// Mitsubishi GX Works2 project: ducthanh   PLC: FX2N/FX2NC

PROGRAM MAIN
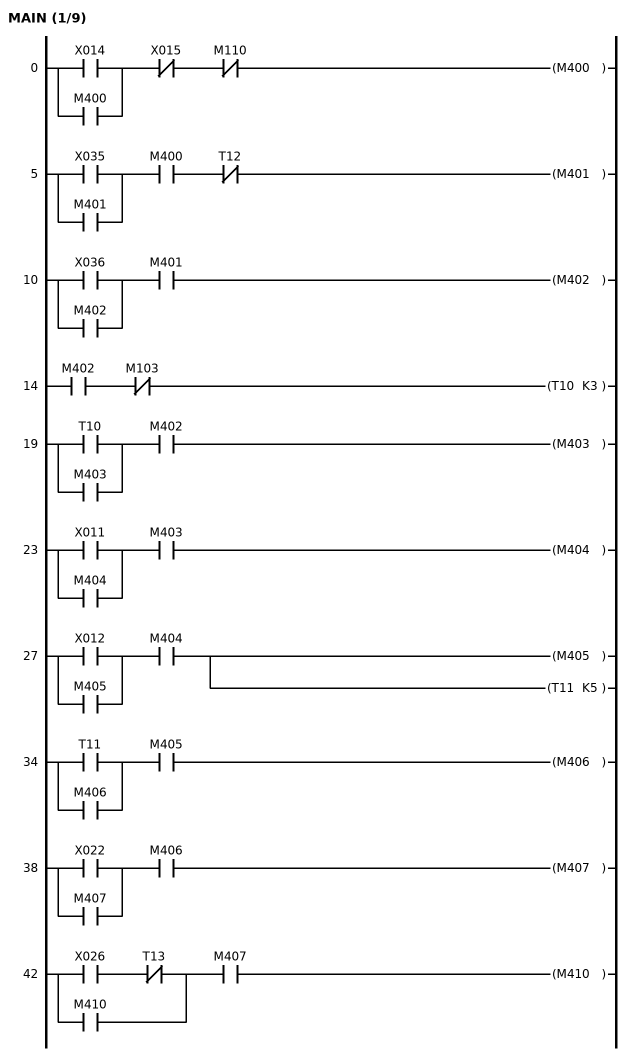
0     LD      X014
      OR      M400
      ANI     X015
      ANI     M110
      OUT     M400
5     LD      X035
      OR      M401
      AND     M400
      ANI     T12
      OUT     M401
10    LD      X036
      OR      M402
      AND     M401
      OUT     M402
14    LD      M402
      ANI     M103
      OUT     T10 K3
19    LD      T10
      OR      M403
      AND     M402
      OUT     M403
23    LD      X011
      OR      M404
      AND     M403
      OUT     M404
27    LD      X012
      OR      M405
      AND     M404
      OUT     M405
      OUT     T11 K5
34    LD      T11
      OR      M406
      AND     M405
      OUT     M406
38    LD      X022
      OR      M407
      AND     M406
      OUT     M407
42    LD      X026
      ANI     T13
      OR      M410
      AND     M407
      OUT     M410
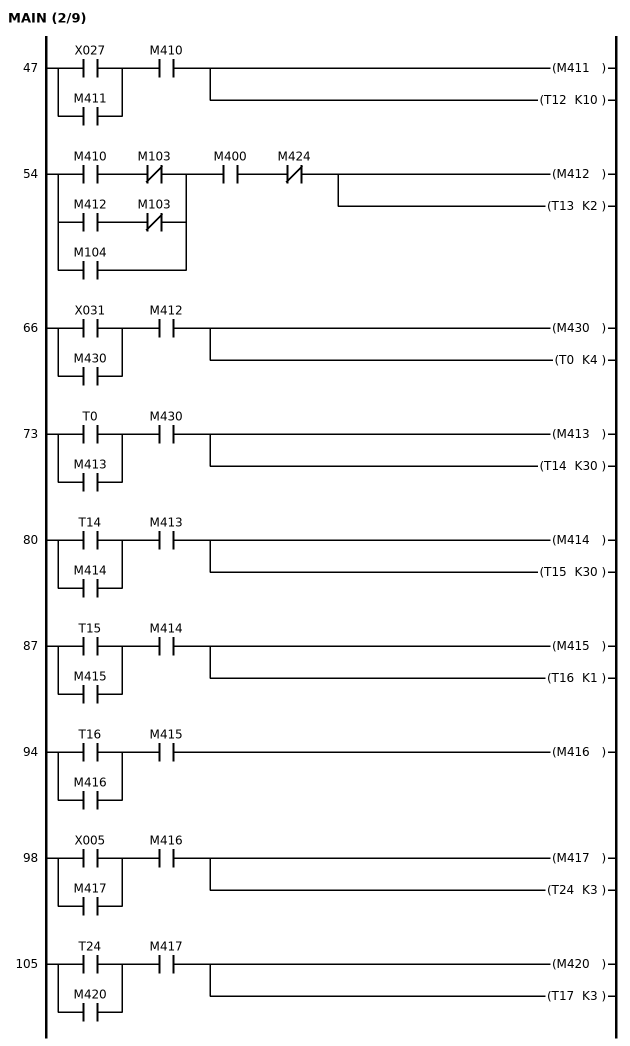
47    LD      X027
      OR      M411
      AND     M410
      OUT     M411
      OUT     T12 K10
54    LD      M410
      ANI     M103
      LD      M412
      ANI     M103
      ORB
      OR      M104
      AND     M400
      ANI     M424
      OUT     M412
      OUT     T13 K2
66    LD      X031
      OR      M430
      AND     M412
      OUT     M430
      OUT     T0 K4
73    LD      T0
      OR      M413
      AND     M430
      OUT     M413
      OUT     T14 K30
80    LD      T14
      OR      M414
      AND     M413
      OUT     M414
      OUT     T15 K30
87    LD      T15
      OR      M415
      AND     M414
      OUT     M415
      OUT     T16 K1
94    LD      T16
      OR      M416
      AND     M415
      OUT     M416
98    LD      X005
      OR      M417
      AND     M416
      OUT     M417
      OUT     T24 K3
105   LD      T24
      OR      M420
      AND     M417
      OUT     M420
      OUT     T17 K3
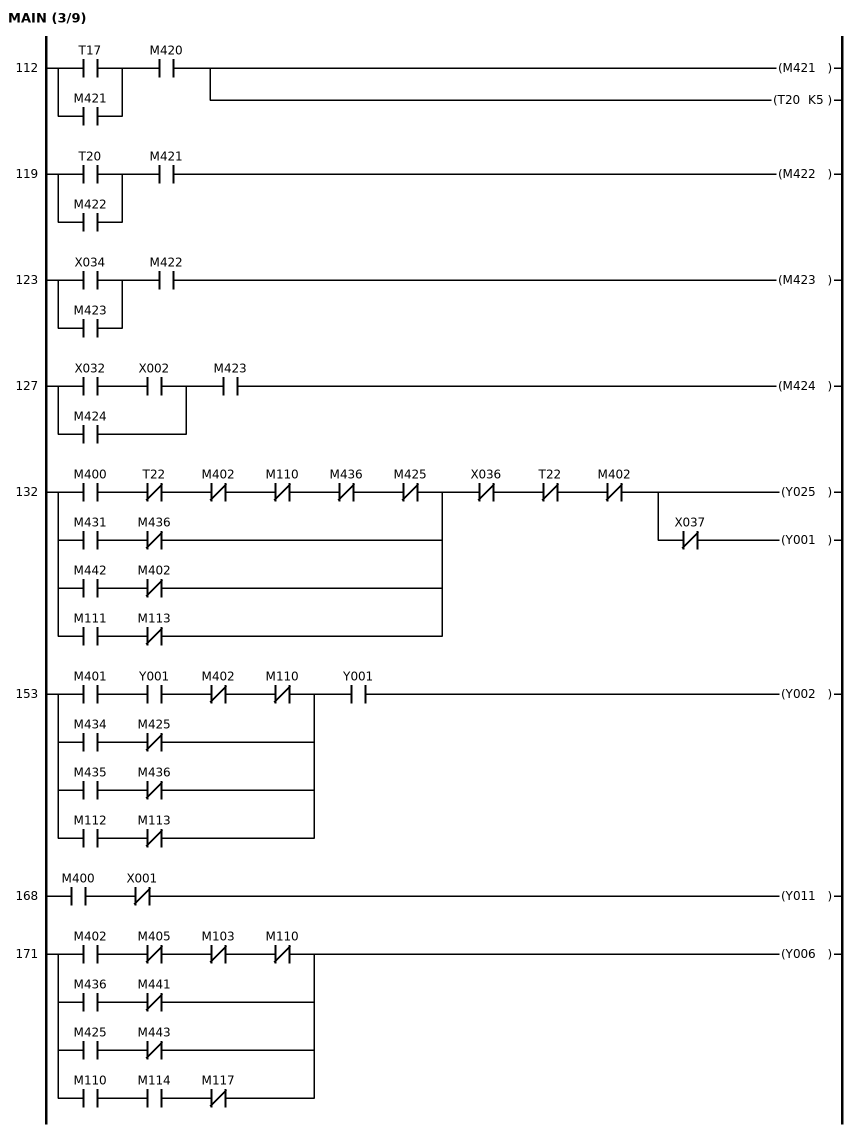
112   LD      T17
      OR      M421
      AND     M420
      OUT     M421
      OUT     T20 K5
119   LD      T20
      OR      M422
      AND     M421
      OUT     M422
123   LD      X034
      OR      M423
      AND     M422
      OUT     M423
127   LD      X032
      AND     X002
      OR      M424
      AND     M423
      OUT     M424
132   LD      M400
      ANI     T22
      ANI     M402
      ANI     M110
      ANI     M436
      ANI     M425
      LD      M431
      ANI     M436
      ORB
      LD      M442
      ANI     M402
      ORB
      LD      M111
      ANI     M113
      ORB
      ANI     X036
      ANI     T22
      ANI     M402
      OUT     Y025
      ANI     X037
      OUT     Y001
153   LD      M401
      AND     Y001
      ANI     M402
      ANI     M110
      LD      M434
      ANI     M425
      ORB
      LD      M435
      ANI     M436
      ORB
      LD      M112
      ANI     M113
      ORB
      AND     Y001
      OUT     Y002
168   LD      M400
      ANI     X001
      OUT     Y011
171   LD      M402
      ANI     M405
      ANI     M103
      ANI     M110
      LD      M436
      ANI     M441
      ORB
      LD      M425
      ANI     M443
      ORB
      LD      M110
      AND     M114
      ANI     M117
      ORB
      OUT     Y006
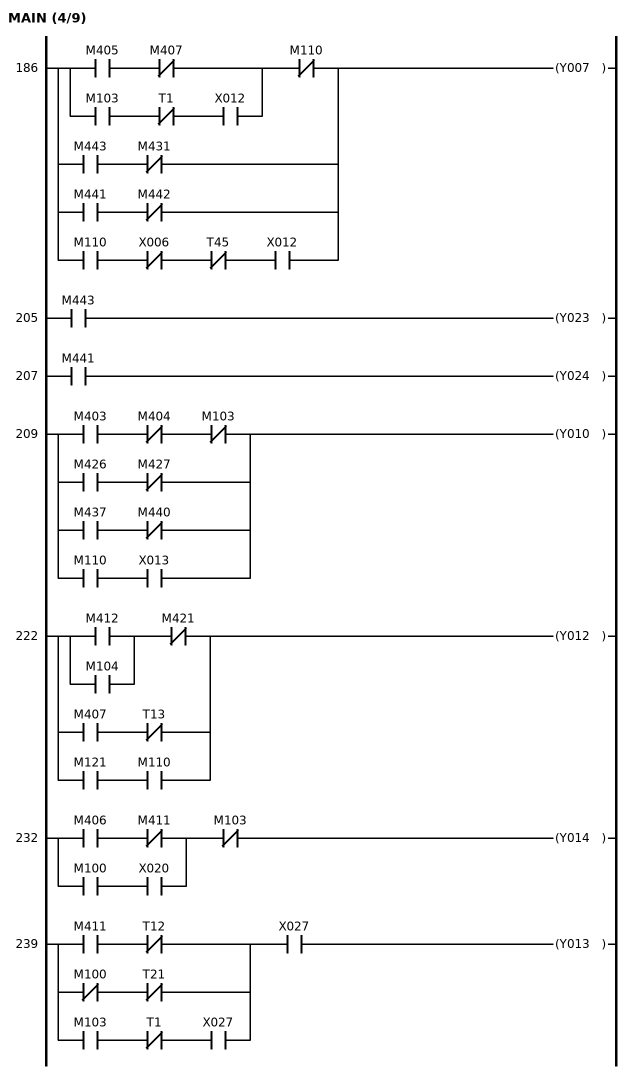
186   LD      M405
      ANI     M407
      LD      M103
      ANI     T1
      AND     X012
      ORB
      ANI     M110
      LD      M443
      ANI     M431
      ORB
      LD      M441
      ANI     M442
      ORB
      LD      M110
      ANI     X006
      ANI     T45
      AND     X012
      ORB
      OUT     Y007
205   LD      M443
      OUT     Y023
207   LD      M441
      OUT     Y024
209   LD      M403
      ANI     M404
      ANI     M103
      LD      M426
      ANI     M427
      ORB
      LD      M437
      ANI     M440
      ORB
      LD      M110
      AND     X013
      ORB
      OUT     Y010
222   LD      M412
      OR      M104
      ANI     M421
      LD      M407
      ANI     T13
      ORB
      LD      M121
      AND     M110
      ORB
      OUT     Y012
232   LD      M406
      ANI     M411
      LD      M100
      AND     X020
      ORB
      ANI     M103
      OUT     Y014
239   LD      M411
      ANI     T12
      LDI     M100
      ANI     T21
      ORB
      LD      M103
      ANI     T1
      AND     X027
      ORB
      AND     X027
      OUT     Y013
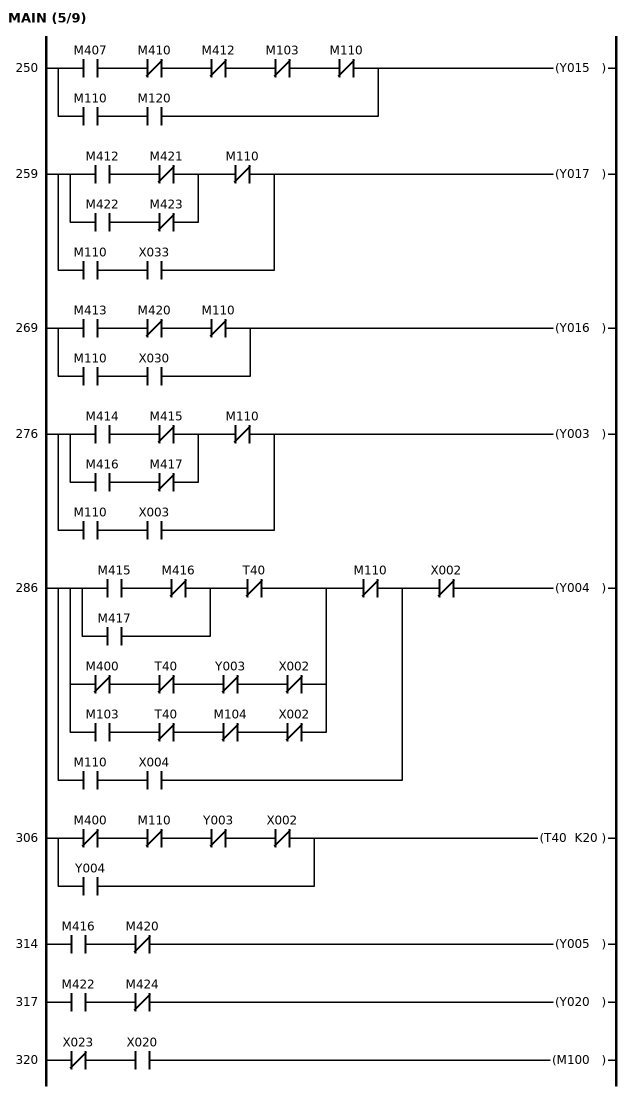
250   LD      M407
      ANI     M410
      ANI     M412
      ANI     M103
      ANI     M110
      LD      M110
      AND     M120
      ORB
      OUT     Y015
259   LD      M412
      ANI     M421
      LD      M422
      ANI     M423
      ORB
      ANI     M110
      LD      M110
      AND     X033
      ORB
      OUT     Y017
269   LD      M413
      ANI     M420
      ANI     M110
      LD      M110
      AND     X030
      ORB
      OUT     Y016
276   LD      M414
      ANI     M415
      LD      M416
      ANI     M417
      ORB
      ANI     M110
      LD      M110
      AND     X003
      ORB
      OUT     Y003
286   LD      M415
      ANI     M416
      OR      M417
      ANI     T40
      LDI     M400
      ANI     T40
      ANI     Y003
      ANI     X002
      ORB
      LD      M103
      ANI     T40
      ANI     M104
      ANI     X002
      ORB
      ANI     M110
      LD      M110
      AND     X004
      ORB
      ANI     X002
      OUT     Y004
306   LDI     M400
      ANI     M110
      ANI     Y003
      ANI     X002
      OR      Y004
      OUT     T40 K20
314   LD      M416
      ANI     M420
      OUT     Y005
317   LD      M422
      ANI     M424
      OUT     Y020
320   LDI     X023
      AND     X020
      OUT     M100
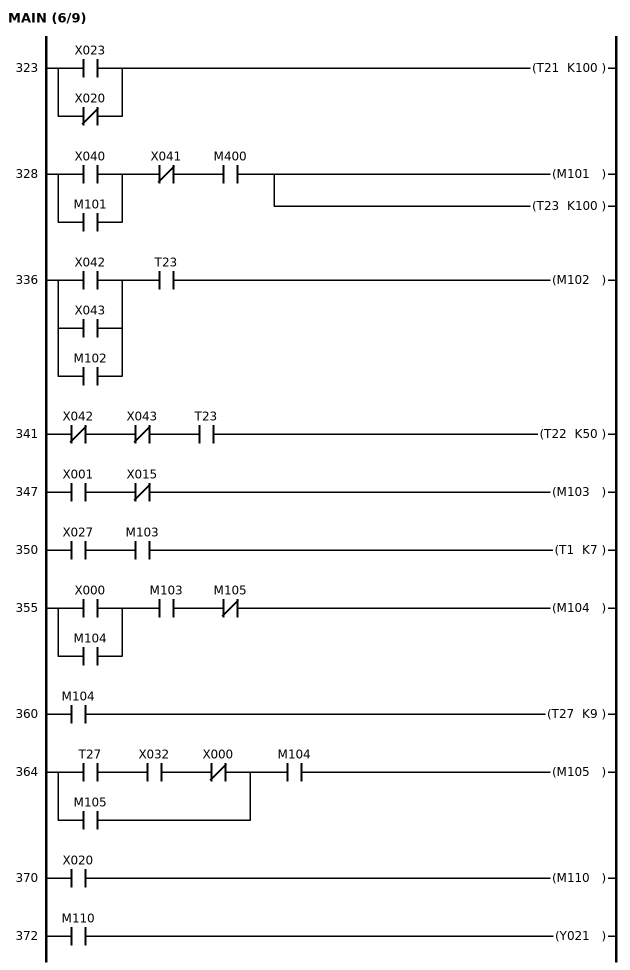
323   LD      X023
      ORI     X020
      OUT     T21 K100
328   LD      X040
      OR      M101
      ANI     X041
      AND     M400
      OUT     M101
      OUT     T23 K100
336   LD      X042
      OR      X043
      OR      M102
      AND     T23
      OUT     M102
341   LDI     X042
      ANI     X043
      AND     T23
      OUT     T22 K50
347   LD      X001
      ANI     X015
      OUT     M103
350   LD      X027
      AND     M103
      OUT     T1 K7
355   LD      X000
      OR      M104
      AND     M103
      ANI     M105
      OUT     M104
360   LD      M104
      OUT     T27 K9
364   LD      T27
      AND     X032
      ANI     X000
      OR      M105
      AND     M104
      OUT     M105
370   LD      X020
      OUT     M110
372   LD      M110
      OUT     Y021
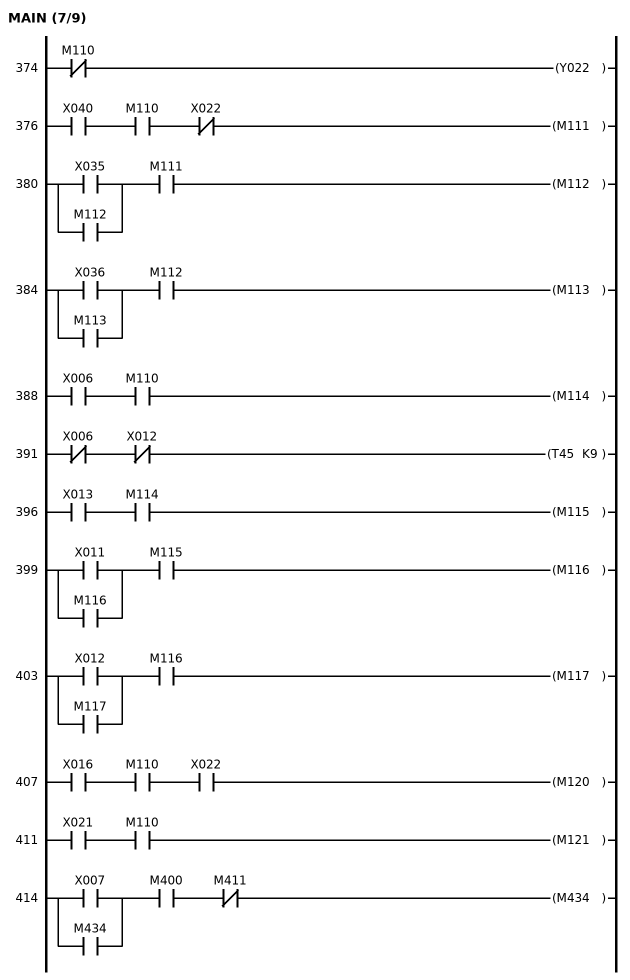
374   LDI     M110
      OUT     Y022
376   LD      X040
      AND     M110
      ANI     X022
      OUT     M111
380   LD      X035
      OR      M112
      AND     M111
      OUT     M112
384   LD      X036
      OR      M113
      AND     M112
      OUT     M113
388   LD      X006
      AND     M110
      OUT     M114
391   LDI     X006
      ANI     X012
      OUT     T45 K9
396   LD      X013
      AND     M114
      OUT     M115
399   LD      X011
      OR      M116
      AND     M115
      OUT     M116
403   LD      X012
      OR      M117
      AND     M116
      OUT     M117
407   LD      X016
      AND     M110
      AND     X022
      OUT     M120
411   LD      X021
      AND     M110
      OUT     M121
414   LD      X007
      OR      M434
      AND     M400
      ANI     M411
      OUT     M434
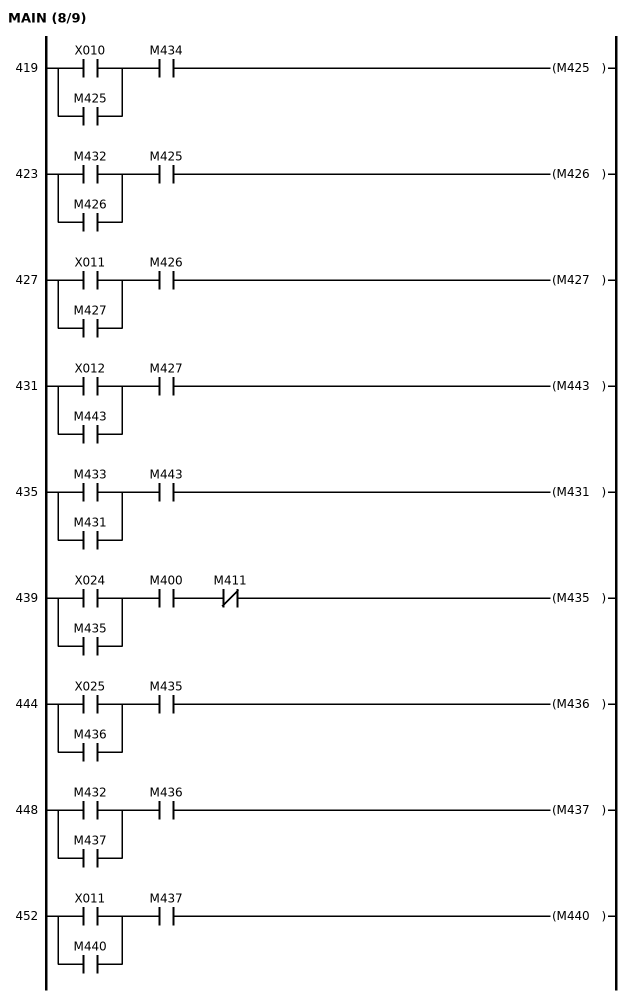
419   LD      X010
      OR      M425
      AND     M434
      OUT     M425
423   LD      M432
      OR      M426
      AND     M425
      OUT     M426
427   LD      X011
      OR      M427
      AND     M426
      OUT     M427
431   LD      X012
      OR      M443
      AND     M427
      OUT     M443
435   LD      M433
      OR      M431
      AND     M443
      OUT     M431
439   LD      X024
      OR      M435
      AND     M400
      ANI     M411
      OUT     M435
444   LD      X025
      OR      M436
      AND     M435
      OUT     M436
448   LD      M432
      OR      M437
      AND     M436
      OUT     M437
452   LD      X011
      OR      M440
      AND     M437
      OUT     M440
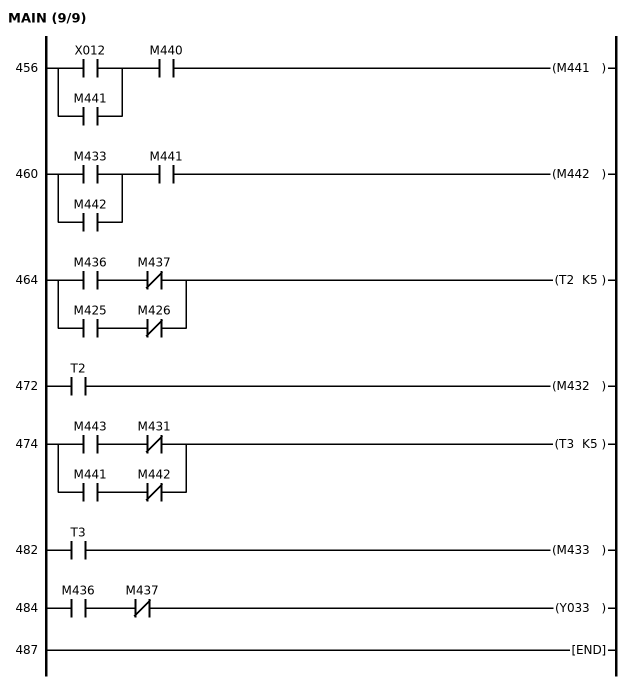
456   LD      X012
      OR      M441
      AND     M440
      OUT     M441
460   LD      M433
      OR      M442
      AND     M441
      OUT     M442
464   LD      M436
      ANI     M437
      LD      M425
      ANI     M426
      ORB
      OUT     T2 K5
472   LD      T2
      OUT     M432
474   LD      M443
      ANI     M431
      LD      M441
      ANI     M442
      ORB
      OUT     T3 K5
482   LD      T3
      OUT     M433
484   LD      M436
      ANI     M437
      OUT     Y033
487   END
END_PROGRAM
